// TIA Portal V17 export
// export: Created 2025-05-22T06:01:57.4466338Z, ExportSetting WithDefaults, DisplayName Totally Integrated Automation Portal, DisplayVersion V17 Update 8, DisplayName TIA Portal Openness, DisplayVersion V17 Update 8, DisplayName TIA Portal Version Control Interface, DisplayVersion V17, DisplayName SINAMICS Startdrive Advanced, DisplayVersion V17 SP2, DisplayName SINAMICS Startdrive G110M, G120, G120C, G120D, G120P, G115D, DisplayVersion V17 SP2, DisplayName SINAMICS Startdrive G130, G150, S120, S150, SINAMICS MV, S210, DisplayVersion V17 SP2, DisplayName STEP 7 Professional, DisplayVersion V17 Update 8, DisplayName SINUMERIK ONE STEP 7 Toolbox, DisplayVersion V17 Update 12, DisplayName SINUMERIK ONE PLC Basic Program Plus, DisplayVersion V17 Update 12, DisplayName SINUMERIK 840D sl STEP 7 Toolbox, DisplayVersion V17 Update 12, DisplayName STEP 7 Safety, DisplayVersion V17 Update 6, DisplayName WinCC Advanced, DisplayVersion V17 Update 8
DATA_BLOCK "DB16304_METHODCALL_U1_STA3_MEAS_MEAS_LAYER_STOP_CON_MGR"   // DB16304
{ DB_Accessible_From_OPC_UA := 'FALSE' }
VERSION : 0.1
// stored: AutoNumber false, DBAccessibleFromOPCUA false, DBAccessibleFromWebserver false, InstanceOfName FB16001_METHODS_CONNECTION_MGR, InstanceOfType FB
"FB16001_METHODS_CONNECTION_MGR"
   // VAR_INPUT
   //    METHOD_DONE : Bool;
   //    METHOD_ERROR : Bool;
   //    METHOD_BUSY : Bool;
   //    METHOD_STATUS : DWord;
   //    OPC_UA_Connect : DWord;
   //    OPC_UA_NamespaceGetIndexList : DWord;
   //    OPC_UA_MethodGetHandleList : DWord;
   //    OPC_UA_MethodCall : DWord;
   //    OPC_UA_MethodReleaseHandleList : DWord;
   //    OPC_UA_Disconnect : DWord;
   //    OPC_UA_ConnectionGetStatus : DWord;
   //    MAX_CON_ATTEMPTS : Int;
   // END_VAR
   // VAR_OUTPUT
   //    RETRY : Bool;
   //    CONNECTION_ERROR : Bool;
   //    CONNECTION_ERROR_STATUS : "CONNECTION_ERROR_STATUS";
   // END_VAR
   // VAR
   //    LAST_ERROR_TIME_STAMP : DTL;
   //    ERROR_FROM_METHOD : Bool;
   //    ERROR_COUNTER : Int;
   //    AUX_PULSE : Bool;
   //    AUX_PULSE_1 : Bool;
   //    AUX_PULSE_2 : Bool;
   //    ZERO : Int;
   //    RET_VAL : Int;
   // END_VAR
BEGIN
END_DATA_BLOCK
